# EPICS IOC start-up script: vme_iocs/iocbio4/iocBoot/st_SIS3820.iocsh
epicsEnvSet("PREFIX",                   "18ID:mcs:")
epicsEnvSet("RNAME",                    "mca")
epicsEnvSet("MAX_SIGNALS",              "32")
epicsEnvSet("MAX_CHANS",                "15000")
epicsEnvSet("PORT",                     "SIS3820/1")
# For MCA records FIELD=READ, for waveform records FIELD=PROC
epicsEnvSet("FIELD",                    "READ")
epicsEnvSet("MODEL",                    "SIS3820")

#drvSIS3820Config("Port name",
#                  baseAddress,
#                  interruptVector,
#                  int interruptLevel,
#                  channels,
#                  signals,
#                  use DMA
#                  fifoBufferWords)
drvSIS3820Config($(PORT), 0xA0000000, 220, 6, $(MAX_CHANS), $(MAX_SIGNALS), 1, 0x2000)

# Update SIS3820 firmware:
# connect pins 2 and 3 on jumper J570
#sis3820_jtag_prom_epics(0xA8000000, "R", "")
# copy prom_v0111.mcs from $(MCA)/mcaApp/SISSrc
#sis3820_jtag_prom_epics(0xA8000000, "P", "prom_v0111.mcs")
#sis3820_jtag_prom_epics(0xA8000000, "V", "prom_v0111.mcs")
# connect pins 1 and 2 on jumper J570

# This loads the scaler record and supporting records
dbLoadRecords("$(STD)/stdApp/Db/scaler32.db", "P=$(PREFIX), S=scaler1, DTYP=Asyn Scaler, OUT=@asyn($(PORT)), FREQ=50000000")

# This database provides the support for the MCS functions
dbLoadRecords("$(MCA)/mcaApp/Db/SIS38XX.template", "P=$(PREFIX), PORT=$(PORT), SCALER=$(PREFIX)scaler1")
# This SNL programs reads the MCS
doAfterIocInit("seq(&SIS38XX_SNL, 'P=$(PREFIX), R=$(RNAME), NUM_SIGNALS=$(MAX_SIGNALS), FIELD=READ')")

# Load either MCA or waveform records below
# The number of records loaded must be the same as MAX_SIGNALS defined above

# Load the MCA records
dbLoadRecords("$(MCA)/mcaApp/Db/simple_mca.db", "P=$(PREFIX), M=$(RNAME)1,  DTYP=asynMCA, INP=@asyn($(PORT) 0),  PREC=3, CHANS=$(MAX_CHANS)")
dbLoadRecords("$(MCA)/mcaApp/Db/simple_mca.db", "P=$(PREFIX), M=$(RNAME)2,  DTYP=asynMCA, INP=@asyn($(PORT) 1),  PREC=3, CHANS=$(MAX_CHANS)")
dbLoadRecords("$(MCA)/mcaApp/Db/simple_mca.db", "P=$(PREFIX), M=$(RNAME)3,  DTYP=asynMCA, INP=@asyn($(PORT) 2),  PREC=3, CHANS=$(MAX_CHANS)")
dbLoadRecords("$(MCA)/mcaApp/Db/simple_mca.db", "P=$(PREFIX), M=$(RNAME)4,  DTYP=asynMCA, INP=@asyn($(PORT) 3),  PREC=3, CHANS=$(MAX_CHANS)")
dbLoadRecords("$(MCA)/mcaApp/Db/simple_mca.db", "P=$(PREFIX), M=$(RNAME)5,  DTYP=asynMCA, INP=@asyn($(PORT) 4),  PREC=3, CHANS=$(MAX_CHANS)")
dbLoadRecords("$(MCA)/mcaApp/Db/simple_mca.db", "P=$(PREFIX), M=$(RNAME)6,  DTYP=asynMCA, INP=@asyn($(PORT) 5),  PREC=3, CHANS=$(MAX_CHANS)")
dbLoadRecords("$(MCA)/mcaApp/Db/simple_mca.db", "P=$(PREFIX), M=$(RNAME)7,  DTYP=asynMCA, INP=@asyn($(PORT) 6),  PREC=3, CHANS=$(MAX_CHANS)")
dbLoadRecords("$(MCA)/mcaApp/Db/simple_mca.db", "P=$(PREFIX), M=$(RNAME)8,  DTYP=asynMCA, INP=@asyn($(PORT) 7),  PREC=3, CHANS=$(MAX_CHANS)")
dbLoadRecords("$(MCA)/mcaApp/Db/simple_mca.db", "P=$(PREFIX), M=$(RNAME)9,  DTYP=asynMCA, INP=@asyn($(PORT) 8),  PREC=3, CHANS=$(MAX_CHANS)")
dbLoadRecords("$(MCA)/mcaApp/Db/simple_mca.db", "P=$(PREFIX), M=$(RNAME)10, DTYP=asynMCA, INP=@asyn($(PORT) 9),  PREC=3, CHANS=$(MAX_CHANS)")
dbLoadRecords("$(MCA)/mcaApp/Db/simple_mca.db", "P=$(PREFIX), M=$(RNAME)11, DTYP=asynMCA, INP=@asyn($(PORT) 10), PREC=3, CHANS=$(MAX_CHANS)")
dbLoadRecords("$(MCA)/mcaApp/Db/simple_mca.db", "P=$(PREFIX), M=$(RNAME)12, DTYP=asynMCA, INP=@asyn($(PORT) 11), PREC=3, CHANS=$(MAX_CHANS)")
dbLoadRecords("$(MCA)/mcaApp/Db/simple_mca.db", "P=$(PREFIX), M=$(RNAME)13, DTYP=asynMCA, INP=@asyn($(PORT) 12), PREC=3, CHANS=$(MAX_CHANS)")
dbLoadRecords("$(MCA)/mcaApp/Db/simple_mca.db", "P=$(PREFIX), M=$(RNAME)14, DTYP=asynMCA, INP=@asyn($(PORT) 13), PREC=3, CHANS=$(MAX_CHANS)")
dbLoadRecords("$(MCA)/mcaApp/Db/simple_mca.db", "P=$(PREFIX), M=$(RNAME)15, DTYP=asynMCA, INP=@asyn($(PORT) 14), PREC=3, CHANS=$(MAX_CHANS)")
dbLoadRecords("$(MCA)/mcaApp/Db/simple_mca.db", "P=$(PREFIX), M=$(RNAME)16, DTYP=asynMCA, INP=@asyn($(PORT) 15), PREC=3, CHANS=$(MAX_CHANS)")
dbLoadRecords("$(MCA)/mcaApp/Db/simple_mca.db", "P=$(PREFIX), M=$(RNAME)17, DTYP=asynMCA, INP=@asyn($(PORT) 16), PREC=3, CHANS=$(MAX_CHANS)")
dbLoadRecords("$(MCA)/mcaApp/Db/simple_mca.db", "P=$(PREFIX), M=$(RNAME)18, DTYP=asynMCA, INP=@asyn($(PORT) 17), PREC=3, CHANS=$(MAX_CHANS)")
dbLoadRecords("$(MCA)/mcaApp/Db/simple_mca.db", "P=$(PREFIX), M=$(RNAME)19, DTYP=asynMCA, INP=@asyn($(PORT) 18), PREC=3, CHANS=$(MAX_CHANS)")
dbLoadRecords("$(MCA)/mcaApp/Db/simple_mca.db", "P=$(PREFIX), M=$(RNAME)20, DTYP=asynMCA, INP=@asyn($(PORT) 19), PREC=3, CHANS=$(MAX_CHANS)")
dbLoadRecords("$(MCA)/mcaApp/Db/simple_mca.db", "P=$(PREFIX), M=$(RNAME)21, DTYP=asynMCA, INP=@asyn($(PORT) 20), PREC=3, CHANS=$(MAX_CHANS)")
dbLoadRecords("$(MCA)/mcaApp/Db/simple_mca.db", "P=$(PREFIX), M=$(RNAME)22, DTYP=asynMCA, INP=@asyn($(PORT) 21), PREC=3, CHANS=$(MAX_CHANS)")
dbLoadRecords("$(MCA)/mcaApp/Db/simple_mca.db", "P=$(PREFIX), M=$(RNAME)23, DTYP=asynMCA, INP=@asyn($(PORT) 22), PREC=3, CHANS=$(MAX_CHANS)")
dbLoadRecords("$(MCA)/mcaApp/Db/simple_mca.db", "P=$(PREFIX), M=$(RNAME)24, DTYP=asynMCA, INP=@asyn($(PORT) 23), PREC=3, CHANS=$(MAX_CHANS)")
dbLoadRecords("$(MCA)/mcaApp/Db/simple_mca.db", "P=$(PREFIX), M=$(RNAME)25, DTYP=asynMCA, INP=@asyn($(PORT) 24), PREC=3, CHANS=$(MAX_CHANS)")
dbLoadRecords("$(MCA)/mcaApp/Db/simple_mca.db", "P=$(PREFIX), M=$(RNAME)26, DTYP=asynMCA, INP=@asyn($(PORT) 25), PREC=3, CHANS=$(MAX_CHANS)")
dbLoadRecords("$(MCA)/mcaApp/Db/simple_mca.db", "P=$(PREFIX), M=$(RNAME)27, DTYP=asynMCA, INP=@asyn($(PORT) 26), PREC=3, CHANS=$(MAX_CHANS)")
dbLoadRecords("$(MCA)/mcaApp/Db/simple_mca.db", "P=$(PREFIX), M=$(RNAME)28, DTYP=asynMCA, INP=@asyn($(PORT) 27), PREC=3, CHANS=$(MAX_CHANS)")
dbLoadRecords("$(MCA)/mcaApp/Db/simple_mca.db", "P=$(PREFIX), M=$(RNAME)29, DTYP=asynMCA, INP=@asyn($(PORT) 28), PREC=3, CHANS=$(MAX_CHANS)")
dbLoadRecords("$(MCA)/mcaApp/Db/simple_mca.db", "P=$(PREFIX), M=$(RNAME)30, DTYP=asynMCA, INP=@asyn($(PORT) 29), PREC=3, CHANS=$(MAX_CHANS)")
dbLoadRecords("$(MCA)/mcaApp/Db/simple_mca.db", "P=$(PREFIX), M=$(RNAME)31, DTYP=asynMCA, INP=@asyn($(PORT) 30), PREC=3, CHANS=$(MAX_CHANS)")
dbLoadRecords("$(MCA)/mcaApp/Db/simple_mca.db", "P=$(PREFIX), M=$(RNAME)32, DTYP=asynMCA, INP=@asyn($(PORT) 31), PREC=3, CHANS=$(MAX_CHANS)")

## AL:  This loads MX MCS dark current support
dbLoadRecords("mx_mcs.db","P=18ID:mcs:,M=mca1")
dbLoadRecords("mx_mcs.db","P=18ID:mcs:,M=mca2")
dbLoadRecords("mx_mcs.db","P=18ID:mcs:,M=mca3")
dbLoadRecords("mx_mcs.db","P=18ID:mcs:,M=mca4")
dbLoadRecords("mx_mcs.db","P=18ID:mcs:,M=mca5")
dbLoadRecords("mx_mcs.db","P=18ID:mcs:,M=mca6")
dbLoadRecords("mx_mcs.db","P=18ID:mcs:,M=mca7")
dbLoadRecords("mx_mcs.db","P=18ID:mcs:,M=mca8")
dbLoadRecords("mx_mcs.db","P=18ID:mcs:,M=mca9")
dbLoadRecords("mx_mcs.db","P=18ID:mcs:,M=mca10")
dbLoadRecords("mx_mcs.db","P=18ID:mcs:,M=mca11")
dbLoadRecords("mx_mcs.db","P=18ID:mcs:,M=mca12")
dbLoadRecords("mx_mcs.db","P=18ID:mcs:,M=mca13")
dbLoadRecords("mx_mcs.db","P=18ID:mcs:,M=mca14")
dbLoadRecords("mx_mcs.db","P=18ID:mcs:,M=mca15")
dbLoadRecords("mx_mcs.db","P=18ID:mcs:,M=mca16")
dbLoadRecords("mx_mcs.db","P=18ID:mcs:,M=mca17")
dbLoadRecords("mx_mcs.db","P=18ID:mcs:,M=mca18")
dbLoadRecords("mx_mcs.db","P=18ID:mcs:,M=mca19")
dbLoadRecords("mx_mcs.db","P=18ID:mcs:,M=mca20")
dbLoadRecords("mx_mcs.db","P=18ID:mcs:,M=mca21")
dbLoadRecords("mx_mcs.db","P=18ID:mcs:,M=mca22")
dbLoadRecords("mx_mcs.db","P=18ID:mcs:,M=mca23")
dbLoadRecords("mx_mcs.db","P=18ID:mcs:,M=mca24")
dbLoadRecords("mx_mcs.db","P=18ID:mcs:,M=mca25")
dbLoadRecords("mx_mcs.db","P=18ID:mcs:,M=mca26")
dbLoadRecords("mx_mcs.db","P=18ID:mcs:,M=mca27")
dbLoadRecords("mx_mcs.db","P=18ID:mcs:,M=mca28")
dbLoadRecords("mx_mcs.db","P=18ID:mcs:,M=mca29")
dbLoadRecords("mx_mcs.db","P=18ID:mcs:,M=mca30")
dbLoadRecords("mx_mcs.db","P=18ID:mcs:,M=mca31")
dbLoadRecords("mx_mcs.db","P=18ID:mcs:,M=mca32")

# This loads the waveform records
#dbLoadRecords("$(MCA)/mcaApp/Db/SIS38XX_waveform.template", "P=$(PREFIX), R=$(RNAME)1,  INP=@asyn($(PORT) 0),  CHANS=$(MAX_CHANS)")
#dbLoadRecords("$(MCA)/mcaApp/Db/SIS38XX_waveform.template", "P=$(PREFIX), R=$(RNAME)2,  INP=@asyn($(PORT) 1),  CHANS=$(MAX_CHANS)")
#dbLoadRecords("$(MCA)/mcaApp/Db/SIS38XX_waveform.template", "P=$(PREFIX), R=$(RNAME)3,  INP=@asyn($(PORT) 2),  CHANS=$(MAX_CHANS)")
#dbLoadRecords("$(MCA)/mcaApp/Db/SIS38XX_waveform.template", "P=$(PREFIX), R=$(RNAME)4,  INP=@asyn($(PORT) 3),  CHANS=$(MAX_CHANS)")
#dbLoadRecords("$(MCA)/mcaApp/Db/SIS38XX_waveform.template", "P=$(PREFIX), R=$(RNAME)5,  INP=@asyn($(PORT) 4),  CHANS=$(MAX_CHANS)")
#dbLoadRecords("$(MCA)/mcaApp/Db/SIS38XX_waveform.template", "P=$(PREFIX), R=$(RNAME)6,  INP=@asyn($(PORT) 5),  CHANS=$(MAX_CHANS)")
#dbLoadRecords("$(MCA)/mcaApp/Db/SIS38XX_waveform.template", "P=$(PREFIX), R=$(RNAME)7,  INP=@asyn($(PORT) 6),  CHANS=$(MAX_CHANS)")
#dbLoadRecords("$(MCA)/mcaApp/Db/SIS38XX_waveform.template", "P=$(PREFIX), R=$(RNAME)8,  INP=@asyn($(PORT) 7),  CHANS=$(MAX_CHANS)")
#dbLoadRecords("$(MCA)/mcaApp/Db/SIS38XX_waveform.template", "P=$(PREFIX), R=$(RNAME)9,  INP=@asyn($(PORT) 8),  CHANS=$(MAX_CHANS)")
#dbLoadRecords("$(MCA)/mcaApp/Db/SIS38XX_waveform.template", "P=$(PREFIX), R=$(RNAME)10, INP=@asyn($(PORT) 9),  CHANS=$(MAX_CHANS)")
#dbLoadRecords("$(MCA)/mcaApp/Db/SIS38XX_waveform.template", "P=$(PREFIX), R=$(RNAME)11, INP=@asyn($(PORT) 10), CHANS=$(MAX_CHANS)")
#dbLoadRecords("$(MCA)/mcaApp/Db/SIS38XX_waveform.template", "P=$(PREFIX), R=$(RNAME)12, INP=@asyn($(PORT) 11), CHANS=$(MAX_CHANS)")
#dbLoadRecords("$(MCA)/mcaApp/Db/SIS38XX_waveform.template", "P=$(PREFIX), R=$(RNAME)13, INP=@asyn($(PORT) 12), CHANS=$(MAX_CHANS)")
#dbLoadRecords("$(MCA)/mcaApp/Db/SIS38XX_waveform.template", "P=$(PREFIX), R=$(RNAME)14, INP=@asyn($(PORT) 13), CHANS=$(MAX_CHANS)")
#dbLoadRecords("$(MCA)/mcaApp/Db/SIS38XX_waveform.template", "P=$(PREFIX), R=$(RNAME)15, INP=@asyn($(PORT) 14), CHANS=$(MAX_CHANS)")
#dbLoadRecords("$(MCA)/mcaApp/Db/SIS38XX_waveform.template", "P=$(PREFIX), R=$(RNAME)16, INP=@asyn($(PORT) 15), CHANS=$(MAX_CHANS)")
#dbLoadRecords("$(MCA)/mcaApp/Db/SIS38XX_waveform.template", "P=$(PREFIX), R=$(RNAME)17, INP=@asyn($(PORT) 16), CHANS=$(MAX_CHANS)")
#dbLoadRecords("$(MCA)/mcaApp/Db/SIS38XX_waveform.template", "P=$(PREFIX), R=$(RNAME)18, INP=@asyn($(PORT) 17), CHANS=$(MAX_CHANS)")
#dbLoadRecords("$(MCA)/mcaApp/Db/SIS38XX_waveform.template", "P=$(PREFIX), R=$(RNAME)19, INP=@asyn($(PORT) 18), CHANS=$(MAX_CHANS)")
#dbLoadRecords("$(MCA)/mcaApp/Db/SIS38XX_waveform.template", "P=$(PREFIX), R=$(RNAME)20, INP=@asyn($(PORT) 19), CHANS=$(MAX_CHANS)")
#dbLoadRecords("$(MCA)/mcaApp/Db/SIS38XX_waveform.template", "P=$(PREFIX), R=$(RNAME)21, INP=@asyn($(PORT) 20), CHANS=$(MAX_CHANS)")
#dbLoadRecords("$(MCA)/mcaApp/Db/SIS38XX_waveform.template", "P=$(PREFIX), R=$(RNAME)22, INP=@asyn($(PORT) 21), CHANS=$(MAX_CHANS)")
#dbLoadRecords("$(MCA)/mcaApp/Db/SIS38XX_waveform.template", "P=$(PREFIX), R=$(RNAME)23, INP=@asyn($(PORT) 22), CHANS=$(MAX_CHANS)")
#dbLoadRecords("$(MCA)/mcaApp/Db/SIS38XX_waveform.template", "P=$(PREFIX), R=$(RNAME)24, INP=@asyn($(PORT) 23), CHANS=$(MAX_CHANS)")
#dbLoadRecords("$(MCA)/mcaApp/Db/SIS38XX_waveform.template", "P=$(PREFIX), R=$(RNAME)25, INP=@asyn($(PORT) 24), CHANS=$(MAX_CHANS)")
#dbLoadRecords("$(MCA)/mcaApp/Db/SIS38XX_waveform.template", "P=$(PREFIX), R=$(RNAME)26, INP=@asyn($(PORT) 25), CHANS=$(MAX_CHANS)")
#dbLoadRecords("$(MCA)/mcaApp/Db/SIS38XX_waveform.template", "P=$(PREFIX), R=$(RNAME)27, INP=@asyn($(PORT) 26), CHANS=$(MAX_CHANS)")
#dbLoadRecords("$(MCA)/mcaApp/Db/SIS38XX_waveform.template", "P=$(PREFIX), R=$(RNAME)28, INP=@asyn($(PORT) 27), CHANS=$(MAX_CHANS)")
#dbLoadRecords("$(MCA)/mcaApp/Db/SIS38XX_waveform.template", "P=$(PREFIX), R=$(RNAME)29, INP=@asyn($(PORT) 28), CHANS=$(MAX_CHANS)")
#dbLoadRecords("$(MCA)/mcaApp/Db/SIS38XX_waveform.template", "P=$(PREFIX), R=$(RNAME)30, INP=@asyn($(PORT) 20), CHANS=$(MAX_CHANS)")
#dbLoadRecords("$(MCA)/mcaApp/Db/SIS38XX_waveform.template", "P=$(PREFIX), R=$(RNAME)31, INP=@asyn($(PORT) 30), CHANS=$(MAX_CHANS)")
#dbLoadRecords("$(MCA)/mcaApp/Db/SIS38XX_waveform.template", "P=$(PREFIX), R=$(RNAME)32, INP=@asyn($(PORT) 31), CHANS=$(MAX_CHANS)")

asynSetTraceIOMask($(PORT),0,2)
#asynSetTraceFile("$(PORT)",0,"$(MODEL).out")
#asynSetTraceMask("$(PORT)",0,0xff)
